PROGRAM Load_Lost_Idle
VAR
END_VAR

IF Shuttle.ReturnToIdleTrigger.Q THEN
	
	IF Shuttle.GrabberLoaded[1] OR Shuttle.GrabberLoadInGrabRange[1] THEN
		
		Shuttle.GrabberWasLoadedIdle[1]		:= TRUE;
	
	ELSE
		
		Shuttle.GrabberWasLoadedIdle[1] 	:= FALSE;
	
	END_IF
	
	IF Shuttle.GrabberLoaded[2] OR Shuttle.GrabberLoadInGrabRange[2] THEN
		
		Shuttle.GrabberWasLoadedIdle[2]		:= TRUE;
	
	ELSE
		
		Shuttle.GrabberWasLoadedIdle[2] 	:= FALSE;
	
	END_IF

END_IF

IF Shuttle.ReturnToIdleTrigger.Q THEN

	IF (Shuttle.GrabberWasLoadedIdle[1] AND Shuttle.GrabberLoaded[1] = FALSE) OR 
		(Shuttle.GrabberWasLoadedIdle[2] AND Shuttle.GrabberLoaded[2] = FALSE) THEN
		
		Shuttle.Grabber_Lost_Load			:= TRUE;
	
	ELSE
		
		Shuttle.Grabber_Lost_Load			:= FALSE;
	
	END_IF

END_IF

IF Otto.EnableAttachment THEN
	
	IF Shuttle.ActiveBays[1] = FALSE THEN
		
		IF Shuttle.GrabberWasLoadedIdle[1] AND Shuttle.GrabberLoaded[1] = FALSE THEN
			
			Shuttle.Grabber_Lost_Load			:= TRUE;
		
		END_IF
	
	END_IF
	
	IF Shuttle.ActiveBays[2] = FALSE THEN
		
		IF Shuttle.GrabberWasLoadedIdle[2] AND Shuttle.GrabberLoaded[2] = FALSE THEN
			
			Shuttle.Grabber_Lost_Load			:= TRUE;
		
		END_IF
	
	END_IF

END_IF

IF Shuttle.Reset THEN
	
	Shuttle.Grabber_Lost_Load	:= FALSE;

END_IF

END_PROGRAM

(* stored: Version 1.1.0.1, ProductVersion 3.1.4024.9
   POU Load_Lost_Idle: Id {c5ca50de-a2d7-49de-8358-25a9dac3fb88}, SpecialFunc None *)
